RoboDK station: RDTSDemo1.rdk

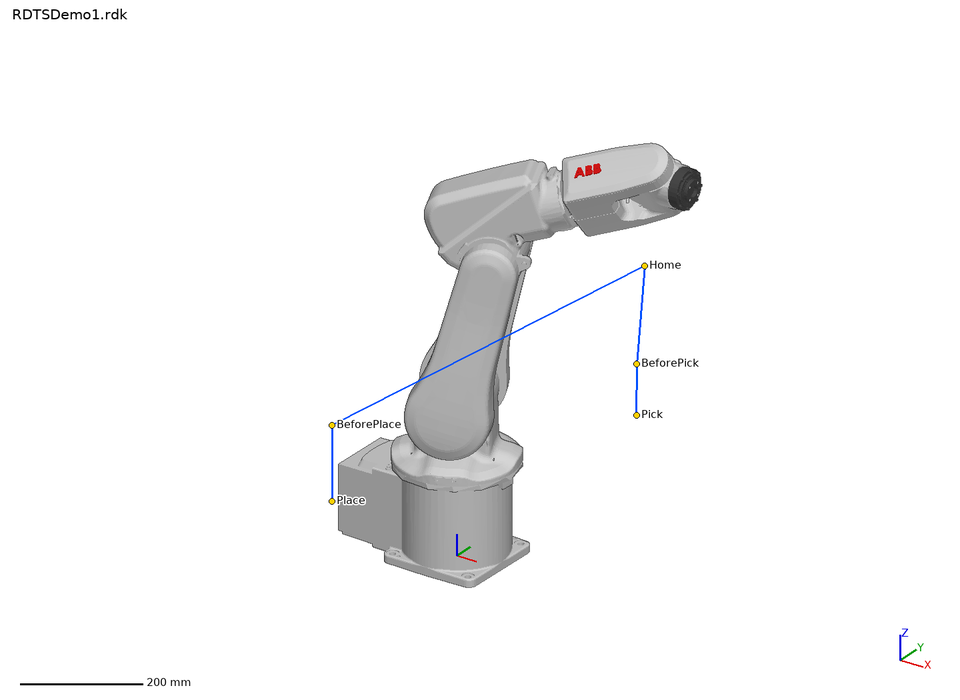
[picture v0: the station drawn from its stored meshes, robots at their saved joint values, targets as dots, program paths as lines]
Station RDTSDemo1 (saved by RoboDK 5.3.2). Poses are relative to the parent item; angles as X-Y-Z fixed-axis rotations.
Station parameters (name, value as stored): 1MoveToPick, 0, 1MakePick, 0, 1PickObjOK, 0, 1MoveToPlace, 1, 1MakePlace, 0, 1PlaceObjOK, 0, 1Waitting, 1
  - frame Robot Base at (0, 0, 0) mm
    - robot Robot (model ABB IRB 120-3/0.6): 6 axes, payload 3 kg, reach 580 mm, repeatability 0.01 mm, weight 25 kg
        modified DH rows (alpha deg, a mm, theta deg, d mm): 0, 0, 0, 290; -90, 0, -90, 0; 0, 270, 0, 0; -90, 70, 0, 302; 90, 0, 0, 0; -90, 0, 180, 72
        joint limits [-165, -110, -90, -160, -120, -400] to [165, 110, 70, 160, 120, 400]; home [0, 0, 0, 0, 0, 0]; saved at [24.81, 14.05, -31.482, -57.055, 30.001, 53.192]
    - target Home (Cartesian target) at (374, 0, 630) mm, rotated rx 0 ry 90 rz 0 deg; joints [0, 0, 0, 0, 0, 0] of Robot
    - target BeforePick (Cartesian target) at (361.4, -4.44, 449.72) mm, rotated rx 179.56 ry -0.69 rz -179.99 deg; joints [-0.79, 11.546, 7.583, 0.457, 71.572, -0.94] of Robot
    - target Pick (Cartesian target) at (360.26, -3.72, 356.24) mm, rotated rx 179.56 ry -0.69 rz -179.99 deg; joints [-0.678, 16.286, 19.725, 0.533, 54.689, -0.992] of Robot
    - target AfterPick (Cartesian target) at (361.4, -4.44, 449.72) mm, rotated rx 179.56 ry -0.69 rz -179.99 deg; joints [-0.79, 11.546, 7.583, 0.457, 71.572, -0.94] of Robot
    - target BeforePlace (Cartesian target) at (-35.63, -303.28, 347.24) mm, rotated rx -180 ry 0.02 rz 89.3 deg; joints [-96.7, 6.034, 33.712, 0, 50.235, -6] of Robot
    - target Place (Cartesian target) at (-35.63, -303.33, 209.09) mm, rotated rx -180 ry 0.02 rz 89.3 deg; joints [-96.7, 26.83, 39.92, 0, 23.23, -6] of Robot
    - target AfterPlace (Cartesian target) at (-35.63, -303.28, 347.24) mm, rotated rx -180 ry 0.02 rz 89.3 deg; joints [-96.7, 6.034, 33.712, 0, 50.235, -6] of Robot
  - program RobotProg (27 instructions, listed below)
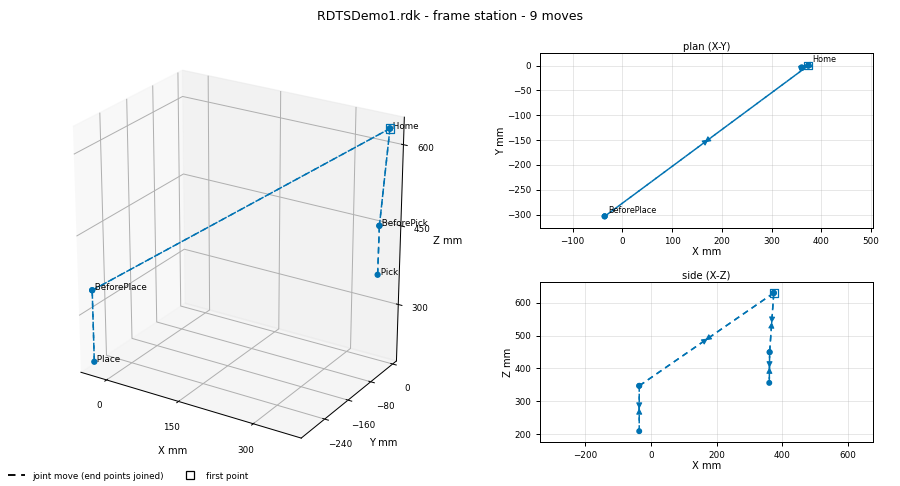
[picture p0: tool path of RDTSDemo1.rdk in frame station, 9 of 9 moves have a stored position in this frame; points joined in program order, loops and branches not executed]

--- program RobotProg (robot Robot) ---
  设置参考: Robot Base
  MoveJ (Home)
  Set 1MakePick=0
  Set 1PickObjOK=0
  Set 1MakePlace=0
  Set 1PlaceObjOK=0
  Wait 1MoveToPick=1
  Set 1Waitting=0
  MoveJ (BeforePick)
  MoveJ (Pick)
  Set 1MakePick=1
  Wait 1PickObjOK=1
  Set 1MakePick=0
  暂停 2.0 s
  MoveJ (AfterPick)
  MoveJ (Home)
  Set 1Waitting=1
  Wait 1MoveToPlace=1
  Set 1Waitting=0
  MoveJ (BeforePlace)
  MoveJ (Place)
  Set 1MakePlace=1
  Wait 1PlaceObjOK=1
  Set 1MakePlace=0
  MoveJ (AfterPlace)
  MoveJ (Home)
  Set 1Waitting=1
